Fanuc KAREL source: ko00067.KL

-- PROVISIONAL review KL for V770-1; original PC SHA256 bbfdd454e24455c3d46e55e6497c396a57d1bf178b8710dcc2842073a0155aa4
-- Incomplete behavior may be omitted. Consult companion uncertainty JSON. Do not deploy.
PROGRAM KO00067
%NOLOCKGROUP
BEGIN
  -- UNRESOLVED_PC offsets 5-12; opcodes 9D,23
  -- UNRESOLVED_PC offsets 17-63; opcodes 27,22,1C,22,1C,22,31,7E,4A
  -- UNRESOLVED_PC offsets 68-72; opcodes 7F
END KO00067
